//////////////////////////////////////////////////////////////////
// Structure For PDL. Main Operating Data to be saved (ex: OPC) //  
//////////////////////////////////////////////////////////////////

TYPE SUBHV :
STRUCT
	// Substation Data
	
	MesAlarmCode				: WORD ; (* (NA) Internal Akuo AlarmCode 	*) 
 	MesWarningCode				: WORD ; (* (NA) Internal Akuo WarningCode  *)
	MesEventCode				: WORD ; (* (NA) Internal Akuo EventCode 	*)
	
END_STRUCT
END_TYPE

(* stored: Version 1.1.0.1, ProductVersion 3.1.4024.6
   DUT SUBHV: Id {9dcd9420-3338-4061-bfc3-9269c1345455} *)
